FUNCTION_BLOCK FB_STATE_MACHINE
VAR_IN_OUT
	State : INT;
	AlarmHandler : FB_ALARM_HANDLER;
END_VAR
VAR_INPUT
	StateAsString : STRING;
	DebugMode : BOOL;
	DebugNext : BOOL;
	StopAllowed : BOOL;
	Timeout : TIME;
END_VAR
VAR_OUTPUT
	CurrentState : INT;
	_firstCycle : BOOL := TRUE;
	StateChangeTime : TIME := TIME();
	Running : BOOL;
	Stopped : BOOL;
	StopRequested : BOOL;
	PreviousState : INT;
END_VAR
VAR
	_changePending : BOOL;
	DelayStart : TIME;
	ChangeDelay : TIME;
	NewState : INT;
	NextState : INT;
	TimeoutAlarm : FB_ALARM;
END_VAR

IF NOT DebugMode THEN
	DebugNext := FALSE;
END_IF;

IF Running AND StopRequested AND StopAllowed THEN
	Running := FALSE;
	Stopped := TRUE;
	StopRequested := FALSE;
END_IF;

IF NewState <> CurrentState AND (NOT DebugMode OR DebugNext) AND Running THEN
	PreviousState := CurrentState;
	CurrentState := NewState;
	StateChangeTime := TIME();
	_firstCycle := TRUE;
	DebugNext := FALSE;
	
	Timeout := T#0S;
	DelayStart := T#0S;
	ChangeDelay := T#0S;
	_changePending := FALSE;
	NextState := 0;
ELSE
	_firstCycle := FALSE;
END_IF;

IF _changePending AND TIME() >= (DelayStart + ChangeDelay) THEN
	THIS^.NewState := NextState;
END_IF;

IF Timeout > T#0S AND THIS^.GetElapsedTime() > Timeout  THEN
	IF NOT TimeoutAlarm.IsActive THEN
		TimeoutAlarm.Config.Name := CONCAT(StateAsString, '*TIMEOUT_ALARM');
		TimeoutAlarm.Activate();
	END_IF;
END_IF;

TimeoutAlarm.Config.Acknowledge := E_ALARM_ACK_TYPE.ONLY_ACK;
TimeoutAlarm.Config.MultiInstance := TRUE;
TimeoutAlarm(Handler := AlarmHandler);

State := CurrentState;

StopAllowed := FALSE;

PROPERTY PUBLIC ChangePending : BOOL
GET
ChangePending := THIS^._changePending;
END_GET
END_PROPERTY

METHOD ChangeState : REFERENCE TO FB_STATE_MACHINE
VAR_INPUT
	State : INT;
END_VAR
IF NOT _changePending AND THIS^.Running THEN
	_changePending := TRUE;
	NextState := State;
END_IF;

ChangeState REF= THIS^;
END_METHOD

METHOD ChangeStateAfterDelay : REFERENCE TO FB_STATE_MACHINE
VAR_INPUT
	State : INT;
	Delay : TIME;
END_VAR
IF NOT _changePending AND THIS^.Running THEN
	_changePending := TRUE;
	NextState := State;
	DelayStart := TIME();
	ChangeDelay := Delay;
END_IF;

ChangeStateAfterDelay REF= THIS^;
END_METHOD

PROPERTY PUBLIC FirstCycle : BOOL
GET
FirstCycle := _firstCycle AND Running;
END_GET
END_PROPERTY

METHOD PUBLIC GetElapsedTime : TIME
VAR_INPUT
END_VAR
GetElapsedTime := TIME() - StateChangeTime;
END_METHOD

METHOD PUBLIC Reset : REFERENCE TO FB_STATE_MACHINE
VAR_INPUT
END_VAR
THIS^.CurrentState := 0;
THIS^.NewState := 0;
THIS^._firstCycle := TRUE;
THIS^.StateChangeTime := TIME();
THIS^._changePending := FALSE;
THIS^.DelayStart := T#0S;
THIS^.ChangeDelay := T#0S;
THIS^.NextState := 0;
THIS^.Running := FALSE;
THIS^.Stopped := FALSE;
THIS^.StopRequested := FALSE;

Reset REF= THIS^;
END_METHOD

{attribute 'TcRpcEnable'}
METHOD PUBLIC Start : REFERENCE TO FB_STATE_MACHINE
VAR_INPUT
END_VAR
THIS^.Running := TRUE;
THIS^.StopRequested := FALSE;

Start REF= THIS^;
END_METHOD

{attribute 'TcRpcEnable'}
METHOD PUBLIC Stop : REFERENCE TO FB_STATE_MACHINE
VAR_INPUT
END_VAR
THIS^.StopRequested := TRUE;

Stop REF= THIS^;
END_METHOD

END_FUNCTION_BLOCK

(* stored: Version 1.1.0.1, ProductVersion 3.1.4024.12
   POU FB_STATE_MACHINE: Id {7d1b6763-e9bf-4251-9730-332ebffa1284}, SpecialFunc None
   Property ChangePending: Id {c3933dbc-44b3-4f8b-8288-0731e877cb96}
   Get Get: Id {08951099-7398-4a3b-81b4-d97920bf8409}
   Method ChangeState: Id {d944d479-1873-42b0-ac26-c88d17df6939}
   Method ChangeStateAfterDelay: Id {8a41a32d-9e87-4d32-8435-d1fe8bc78b79}
   Property FirstCycle: Id {b117b3e9-9958-43f3-bd94-da2b0501908c}
   Get Get: Id {5de37df5-c889-44e7-8dc1-bc128e7a196a}
   Method GetElapsedTime: Id {e06b4974-7005-4897-b5f2-5216723e3ee2}
   Method Reset: Id {a422df67-a07a-44c8-b7d7-825481410d27}
   Method Start: Id {2035f4d6-0d00-4498-8f45-5f2f389a8f06}
   Method Stop: Id {e3a56f71-47af-4e26-878b-563e9ccbf174} *)
